FUNCTION_BLOCK PUBLIC FB_AnalogValue IMPLEMENTS I_Observer
VAR_INPUT
END_VAR
VAR_OUTPUT
END_VAR
VAR
	_nActualValue		: BYTE;
END_VAR

{attribute 'monitoring' := 'call'}
PROPERTY nValue : BYTE
GET
nValue := _nActualValue;
END_GET
END_PROPERTY

METHOD Update
VAR_INPUT
	nNewValue		: BYTE;
END_VAR
_nActualValue := nNewValue;
END_METHOD

END_FUNCTION_BLOCK

(* stored: Version 1.1.0.1, ProductVersion 3.1.4024.11
   POU FB_AnalogValue: Id {33d6d243-fb08-490d-9495-c8eca3289fda}, SpecialFunc None
   Property nValue: Id {a61bde19-c47d-43bf-afc1-3803844d2ff4}
   Get Get: Id {1a940b24-2370-44d0-aa60-57f549af0c9e}
   Method Update: Id {9b5a5192-fb75-4a36-8565-4fb8512337b8} *)
